PROGRAM Q1
VAR
END_VAR

(*
LLD, Ladder Logic Diagram
Each function or state can be put into it's own Network.
These Networks are usually activated while a BOOL is true, and usually sets or resets another BOOL at the end.

Advantages include:
	Easy and quick to learn / implement
	Easy to read
	Graphical logic display rather than text
	
Disadvantages include:
	More intricate operations are a bit tricky to implement
	All Networks are executed concurrently so states must be represented by BOOLs
	

*)

// NETWORK 1

END_PROGRAM

(* stored: Version 1.1.0.1, ProductVersion 3.1.4024.12
   POU Q1: Id {3f8f9ebf-0914-4656-bc61-1a8c52a02cad}, SpecialFunc None *)
